(* CODESYS project RTOS_Kursovaya.project

Project tree, tasks and I/O mapping:
  Device : CODESYS Control Win V3 64, 3S - Smart Software Solutions GmbH, version 3.5.5.20
    application Application
      libraries: Standard, * (System); Util, * (System); Standard64, * (System); VisuDialogs, * (System)
      task MainTask (cyclic, interval t#20ms, priority 1) calls PLC_PRG
      task VISU_TASK (cyclic, interval 100 ms, priority 31) calls VisuElems.Visu_Prg
      program PLC_PRG [FBD]
      visualisation RTOS_Interface
      function block CAR_T [FBD]
      global variables GVL
  text list GlobalTextList
  GlobalImagePool
  5ce3da45-db07-42e7-a21c-a00fff4ed8f6|D:\Mr\Download\Telegram Desktop\image_2018-12-10_23-10-47.png
  5ce3da45-db07-42e7-a21c-a00fff4ed8f6|C:\Users\Mr.Sarayra\Pictures\22_tn.jpg
  5ce3da45-db07-42e7-a21c-a00fff4ed8f6|D:\Mr\Download\Telegram Desktop\photo_2018-12-10_15-35-12.jpg
  5ce3da45-db07-42e7-a21c-a00fff4ed8f6|D:\Mr\Download\Telegram Desktop\Snapchat-1179662295.png
*)

// Device/Application/GVL
VAR_GLOBAL
	passengers_C1: INT := 0;
	baggage_st: BOOL := FALSE;
END_VAR

// Device/Application/PLC_PRG
PROGRAM PLC_PRG
VAR
	Price : REAL;
	Passenger_OUT:INT;
	Passenger_IN:INT;
	Direction:INT;
	Bagagge:BOOL;
	Arrived:BOOL;
	Arriving_time:TIME;
	SendRequest:BOOL;
	AcceptRequest:BOOL;
	suitable_car:BOOL;
	Nsuitable_car:BOOL;
	Car_full:BOOL;
	CAR_T_0: CAR_T;
	Direction_1: INT;
	DirectionPP : INT;
	Baggage_O: BOOL;
	DenyRequest:BOOL;
	IN_RADIUS: TIME;
	Match_car:BOOL;
	nMatch_car:BOOL;
	Car_num:INT;
	Arrived_custom: BOOL;
	Direction_custom: INT;
	TP_0: TP;
	DenyLamp: BOOL;
	AcceptLamp:BOOL;
	TP_1: TP;
	Baggage_MV: BOOL;
	Passenger_C1_Sum: INT;
	TP_2: TP;
	TIME_LL: TIME;
	BLINK_0: BLINK;
	d1_l: BOOL;
	d2_l: BOOL;
	d3_l: BOOL;
	d4_l: BOOL;
	TP_3: TP;
	RS_0: RS;
	Arriving_time_USER: TIME;
END_VAR
VAR // added by the converter: edge detectors and wires of the graphical bodies
    _w1, _w2 : BOOL;
END_VAR

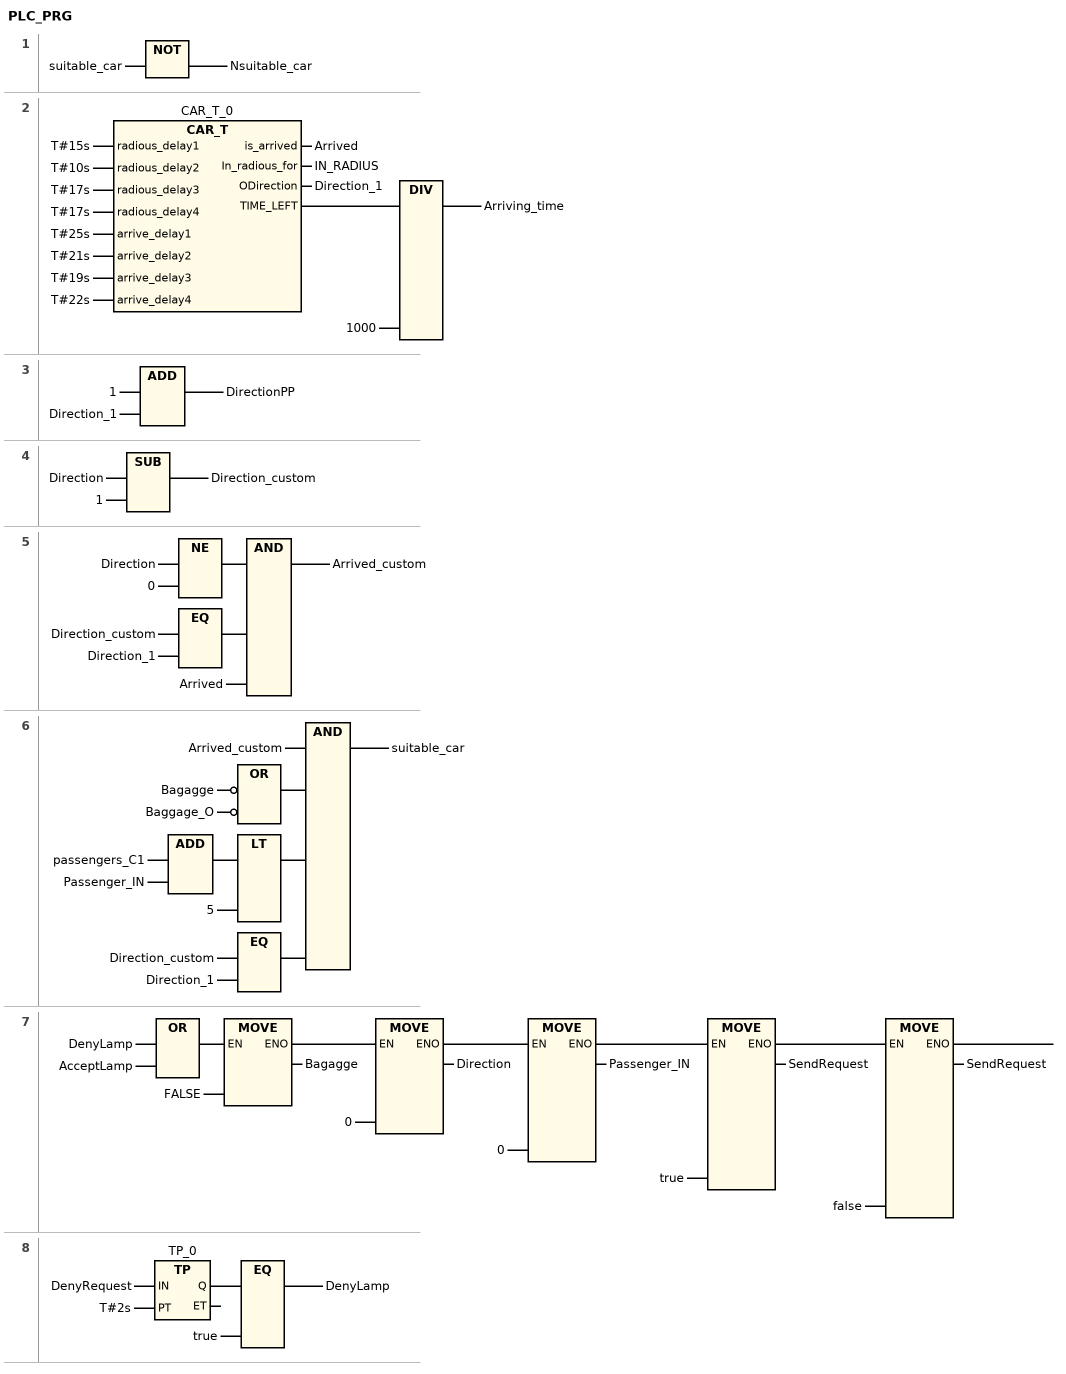
// NETWORK 1
Nsuitable_car := NOT suitable_car;

// NETWORK 2
CAR_T_0(
    radious_delay1 := T#15s,
    radious_delay2 := T#10s,
    radious_delay3 := T#17s,
    radious_delay4 := T#17s,
    arrive_delay1 := T#25s,
    arrive_delay2 := T#21s,
    arrive_delay3 := T#19s,
    arrive_delay4 := T#22s,
    is_arrived => Arrived,
    In_radious_for => IN_RADIUS,
    ODirection => Direction_1); // CAR_T
Arriving_time := CAR_T_0.TIME_LEFT / 1000;

// NETWORK 3
DirectionPP := 1 + Direction_1;

// NETWORK 4
Direction_custom := Direction - 1;

// NETWORK 5
Arrived_custom := Direction <> 0 AND Direction_custom = Direction_1 AND Arrived;

// NETWORK 6
suitable_car := Arrived_custom AND (NOT Bagagge OR NOT Baggage_O) AND passengers_C1 + Passenger_IN < 5 AND Direction_custom = Direction_1;

// NETWORK 7
_w1 := DenyLamp OR AcceptLamp;
IF _w1 THEN Bagagge := FALSE; END_IF
IF _w1 THEN Direction := 0; END_IF
IF _w1 THEN Passenger_IN := 0; END_IF
IF _w1 THEN SendRequest := true; END_IF
IF _w1 THEN SendRequest := false; END_IF

// NETWORK 8
TP_0(IN := DenyRequest, PT := T#2s); // TP
DenyLamp := TP_0.Q = true;

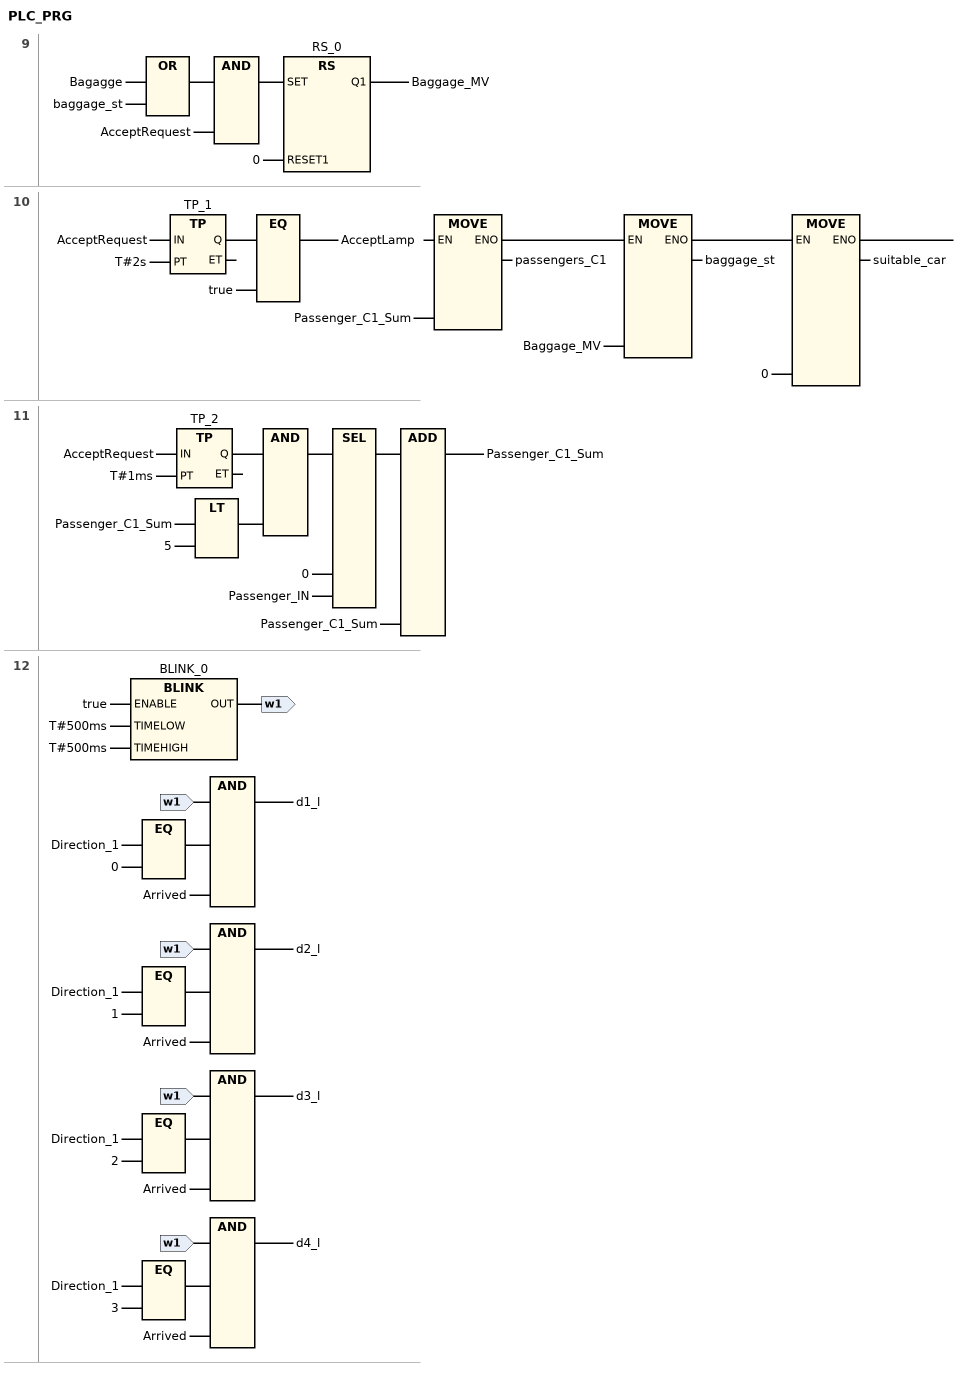
// NETWORK 9
RS_0(SET := (Bagagge OR baggage_st) AND AcceptRequest, RESET1 := 0); // RS
Baggage_MV := RS_0.Q1;

// NETWORK 10
TP_1(IN := AcceptRequest, PT := T#2s); // TP
_w2 := TP_1.Q = true;
AcceptLamp := _w2;
IF _w2 THEN passengers_C1 := Passenger_C1_Sum; END_IF
IF _w2 THEN baggage_st := Baggage_MV; END_IF
IF _w2 THEN suitable_car := 0; END_IF

// NETWORK 11
TP_2(IN := AcceptRequest, PT := T#1ms); // TP
Passenger_C1_Sum := SEL(TP_2.Q AND Passenger_C1_Sum < 5, 0, Passenger_IN) + Passenger_C1_Sum;

// NETWORK 12
BLINK_0(ENABLE := true, TIMELOW := T#500ms, TIMEHIGH := T#500ms); // BLINK
d1_l := BLINK_0.OUT AND Direction_1 = 0 AND Arrived;
d2_l := BLINK_0.OUT AND Direction_1 = 1 AND Arrived;
d3_l := BLINK_0.OUT AND Direction_1 = 2 AND Arrived;
d4_l := BLINK_0.OUT AND Direction_1 = 3 AND Arrived;

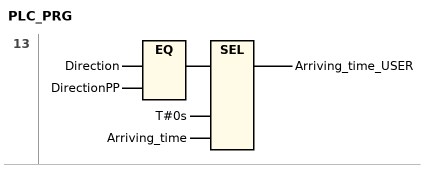
// NETWORK 13
Arriving_time_USER := SEL(Direction = DirectionPP, T#0s, Arriving_time);

END_PROGRAM

// Device/Application/CAR_T
FUNCTION_BLOCK CAR_T
VAR_INPUT


radious_delay1: TIME;
radious_delay2: TIME;
	radious_delay3: TIME;
	radious_delay4: TIME;
	arrive_delay1: TIME;
	arrive_delay2: TIME;
	arrive_delay3: TIME;
	arrive_delay4: TIME;
	
END_VAR
VAR_OUTPUT
	
	is_arrived: BOOL;
	In_radious_for: TIME;
	
	ODirection: WORD;
	TIME_LEFT: TIME;
END_VAR
VAR
	TTT: TIME;
	Arrive_left: TIME;
	In_passengers:INT;
	IN_baggage:BOOL;
	n_arrived: BOOL;
	CTU_0: CTU;
	RESET: BOOL;
	CTU_1: CTU;
	BLINK_1: BLINK;
	Passengers_c: INT;
	TON_0: TON;
	TON_1: TON;
	TP_0: TP;
	TP_1: TP;
	TP_2: TP;
	CTU_2: CTU;
	RESET1: BOOL;
	cycle: WORD;
	temp1: BOOL;
	TOF_0: TOF;

	
END_VAR
VAR // added by the converter: edge detectors and wires of the graphical bodies
    _w1 : BOOL;
END_VAR

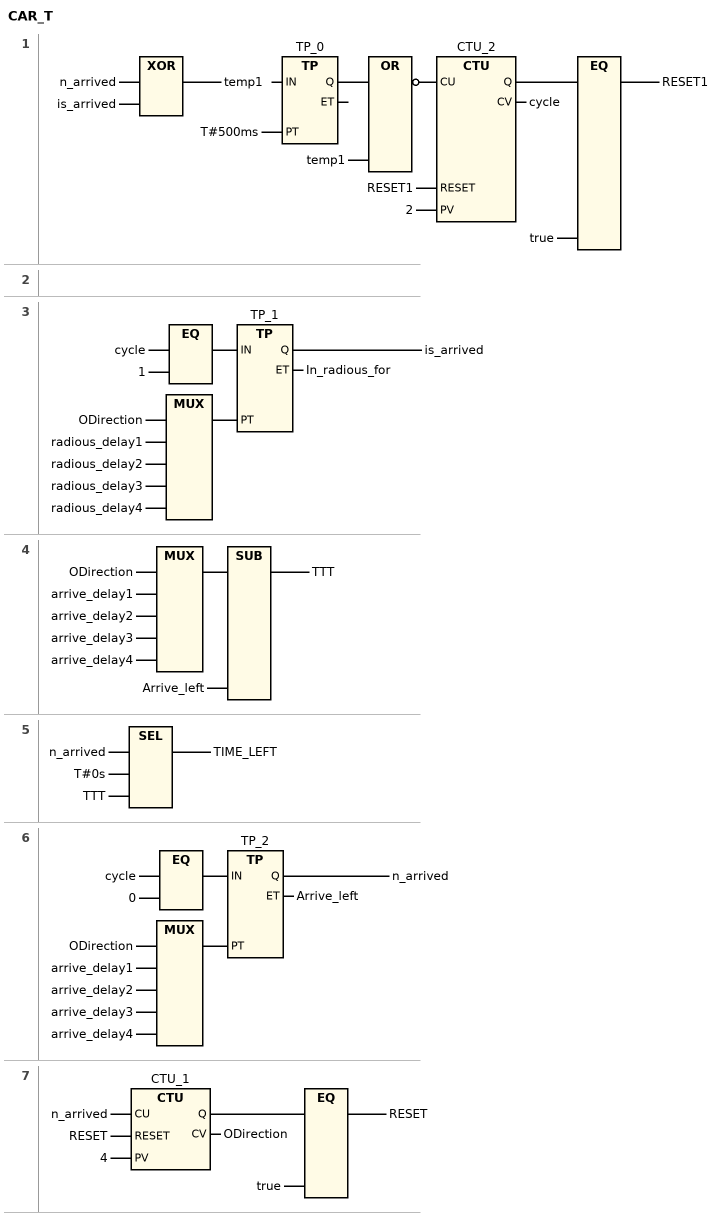
// NETWORK 1
_w1 := n_arrived XOR is_arrived;
temp1 := _w1;
TP_0(IN := _w1, PT := T#500ms); // TP
CTU_2(CU := NOT (TP_0.Q OR temp1), RESET := RESET1, PV := 2, CV => cycle); // CTU
RESET1 := CTU_2.Q = true;

// NETWORK 2

// NETWORK 3
TP_1(
    IN := cycle = 1,
    PT := MUX(ODirection, radious_delay1, radious_delay2, radious_delay3, radious_delay4),
    ET => In_radious_for); // TP
is_arrived := TP_1.Q;

// NETWORK 4
TTT := MUX(ODirection, arrive_delay1, arrive_delay2, arrive_delay3, arrive_delay4) - Arrive_left;

// NETWORK 5
TIME_LEFT := SEL(n_arrived, T#0s, TTT);

// NETWORK 6
TP_2(
    IN := cycle = 0,
    PT := MUX(ODirection, arrive_delay1, arrive_delay2, arrive_delay3, arrive_delay4),
    ET => Arrive_left); // TP
n_arrived := TP_2.Q;

// NETWORK 7
CTU_1(CU := n_arrived, RESET := RESET, PV := 4, CV => ODirection); // CTU
RESET := CTU_1.Q = true;

END_FUNCTION_BLOCK

// Device/Application/RTOS_Interface
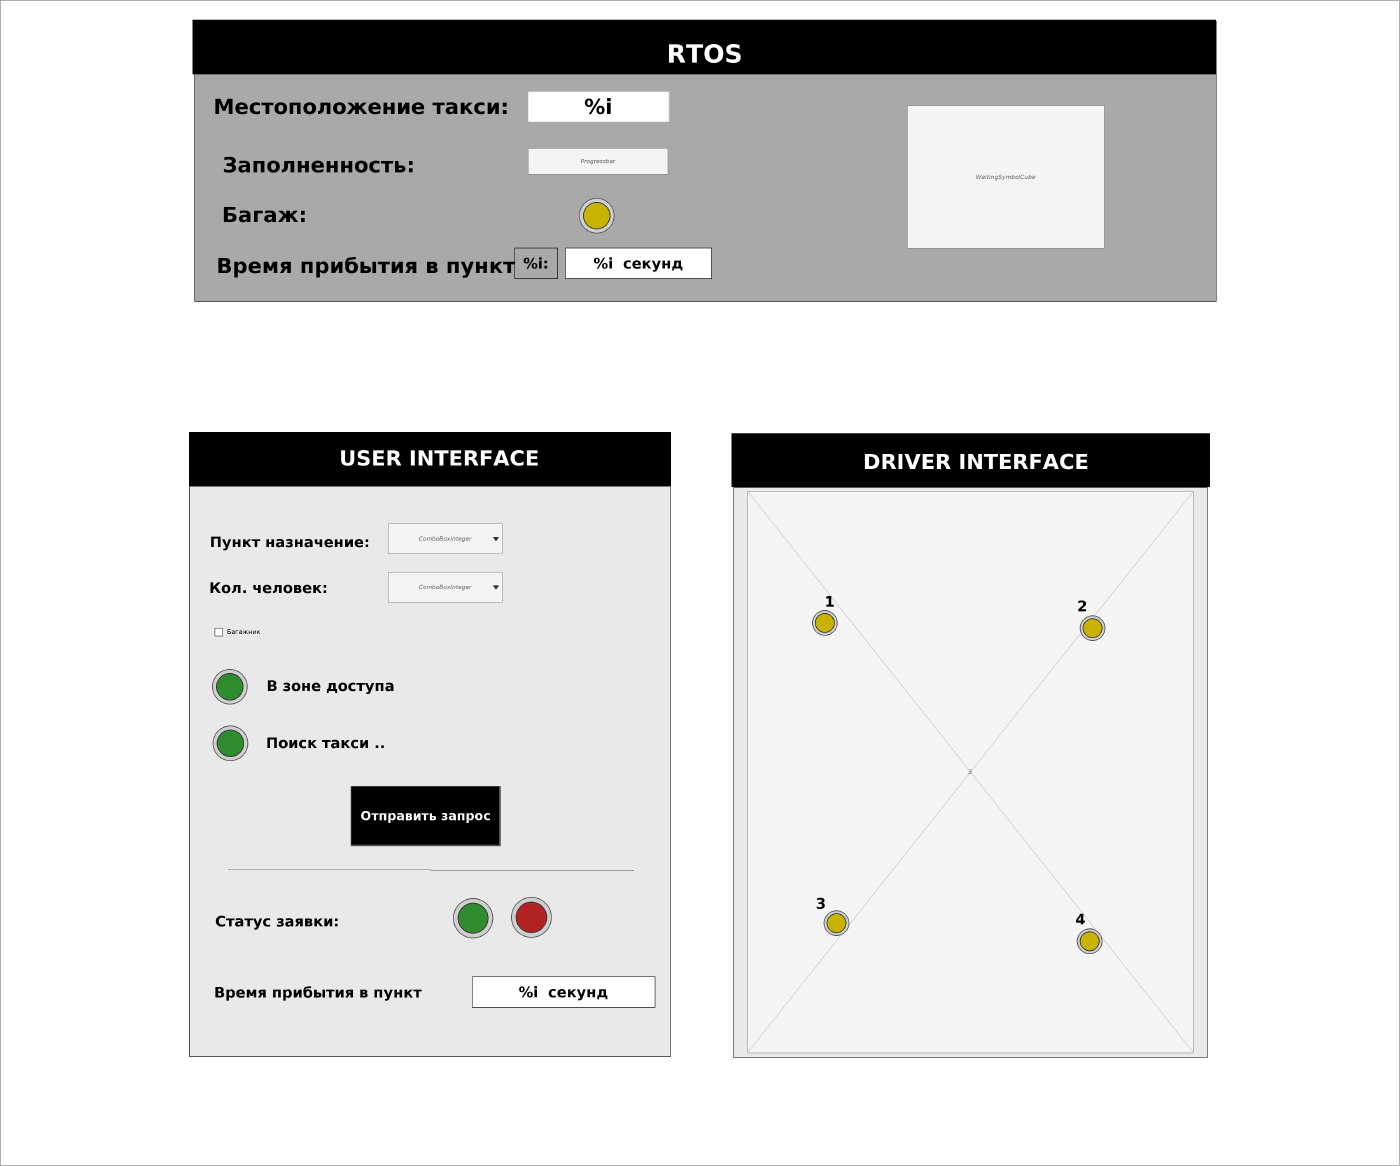
VISUALIZATION RTOS_Interface  // 2400x2000
    Rectangle (333,36 1752x481)
    Rectangle (330,34 1754x93)
    Rectangle (1257,836 813x978), text variable: PLC_PRG.Arriving_time
    Rectangle (1254,743 820x92)
    Label (1469,744 408x96), "DRIVER INTERFACE"
    Textfield (1376,903 588x516)
    Label (1485,934 372x89), "Запрос!"
    Label (1371,1049 372x89), "Кол. пассажиров:"
    Textfield (1847,1063 71x57), "%i", text variable: PLC_PRG.Passenger_IN
    Label (1321,1150 372x89), "Багажник:"
    Lamp1 (1846,1158 70x70), variable: PLC_PRG.Bagagge, style: Lamp-Lamp1-Green
    Button (1723,1448 216x98), "Подтвердить"
        tap PLC_PRG.AcceptRequest
    Button (1410,1449 216x98), "Отклонить"
        tap PLC_PRG.DenyRequest
    Rectangle (324,741 826x92)
    Rectangle (324,834 826x978), text variable: PLC_PRG.Arriving_time
    Label (314,958 293x100), "Кол. человек:"
    Label (350,896 294x67), "Пункт назначение:"
    Checkbox (366,1053 259x62), "Багажник", variable: PLC_PRG.Bagagge
    Lamp1 (359,1143 70x70), variable: PLC_PRG.Arrived_custom, style: Lamp-Lamp1-Green
    Label (391,1128 352x96), "В зоне доступа"
    Label (340,1670 410x64), "Время прибытия в пункт"
    Line (1086,1493) (391,1492)
    Button (601,1348 257x103), "Отправить запрос", invisible if: PLC_PRG.Nsuitable_car
        toggle PLC_PRG.SendRequest
    Textfield (809,1675 314x53), "%i секунд", text variable: PLC_PRG.Arriving_time_USER
    Lamp1 (771,1533 80x84), variable: PLC_PRG.AcceptLamp, style: Lamp-Lamp1-Green
    ComboBoxInteger (665,898 196x52), variable: PLC_PRG.Direction
    ComboBoxInteger (665,981 196x52), variable: PLC_PRG.Passenger_IN
    Lamp1 (360,1240 70x70), variable: PLC_PRG.suitable_car, style: Lamp-Lamp1-Green
    Label (329,1226 459x96), "Поиск такси .."
    Label (577,738 352x96), "USER INTERFACE"
    Lamp1 (867,1533 88x81), variable: PLC_PRG.DenyLamp, style: Lamp-Lamp1-Red
    Label (272,1548 407x64), "Статус заявки:"
    Label (377,153 485x60), "Местоположение такси:"
    Label (908,51 600x83), "RTOS"
    Progressbar (905,254 240x45), variable: passengers_C1
    Label (326,251 441x64), "Заполненность:"
    Textfield (905,157 242x52), "%i", text variable: PLC_PRG.DirectionPP
    WaitingSymbolCube (1555,181 338x245)
    Label (249,318 409x101), "Багаж:"
    Lamp1 (988,335 70x70), variable: baggage_st, style: Lamp-Lamp1-Yellow
    Label (1383,1261 372x89), "Пункт назначение:"
    Textfield (1846,1275 71x57), "%i", text variable: PLC_PRG.Direction
    Image (1281,842 765x964), invisible if: PLC_PRG.SendRequest, image: 3
    Label (1365,1512 85x75), "3", invisible if: PLC_PRG.SendRequest
    Label (1810,1539 85x75), "4", invisible if: PLC_PRG.SendRequest
    Label (1813,1002 85x75), "2", invisible if: PLC_PRG.SendRequest
    Label (1380,994 85x75), "1", invisible if: PLC_PRG.SendRequest
    Lamp1 (1386,1043 56x51), variable: PLC_PRG.d1_l, invisible if: PLC_PRG.SendRequest, style: Lamp-Lamp1-Yellow
    Lamp1 (1845,1052 56x51), variable: PLC_PRG.d2_l, invisible if: PLC_PRG.SendRequest, style: Lamp-Lamp1-Yellow
    Lamp1 (1406,1558 56x51), variable: PLC_PRG.d3_l, invisible if: PLC_PRG.SendRequest, style: Lamp-Lamp1-Yellow
    Lamp1 (1840,1589 56x51), variable: PLC_PRG.d4_l, invisible if: PLC_PRG.SendRequest, style: Lamp-Lamp1-Yellow
    Label (363,424 529x64), "Время прибытия в пункт"
    Textfield (969,425 251x53), "%i секунд", text variable: PLC_PRG.Arriving_time
    Textfield (882,425 74x53), "%i:", text variable: PLC_PRG.DirectionPP
END_VISUALIZATION
